PROGRAM PRG_EncoderSim
VAR
	SimEncoderCount	AT%Q*	:UDINT:=1;	
END_VAR

SimEncoderCount:=SimEncoderCount+1;

IF SimEncoderCount>=4096 THEN
	SimEncoderCount:=1;
END_IF

END_PROGRAM

(* stored: Version 1.1.0.1, ProductVersion 3.1.4024.10
   POU PRG_EncoderSim: Id {8b7b69dd-0b05-4293-8e65-8924344d526a}, SpecialFunc None *)
